TYPE ST_SwitchConfig :
STRUCT
	SwitchCurrent								: INT := 9; //4.0A does crash	
	CurrentMultFactor							: INT 	:= 1310;
	VeloPosnCalcEntry							: LREAL := 0.08;
	VeloPosnCalcExit							: LREAL := 0.06;
	MagnetPosnComp								: LREAL := 100;
	fMagnetEntryPosn 							: LREAL := 10000; //PLEASE ENTER THE MAGNET ENTRY!!!
	fMagnetExitPosn								: LREAL := 10555; //PLEASE ENTER THE MAGNET EXIT!!!
 	SwitchMode        							: E_SwitchOpMode;
	ModeChangeInMotionOK						: BOOL;
	ShuttleCountToDivert						: USINT;
END_STRUCT
END_TYPE;

(* stored: Version 1.1.0.1
   DUT ST_SwitchConfig: Id {1b01e06e-3ad9-017e-0490-e818c7958e80} *)
